FUNCTION_BLOCK FB_CanInterfaceTransport

VAR_INPUT
    bEnable      : BOOL;
END_VAR

VAR_OUTPUT
    xReady       : BOOL;
    xError       : BOOL;
    sErrorText   : STRING(80);
END_VAR

VAR
	TxCanQueue AT%Q* : ST_CanQueue;
	RxCanQueue AT%I* : ST_CanQueue;
END_VAR

END_FUNCTION_BLOCK

(* stored: Version 1.1.0.1
   POU FB_CanInterfaceTransport: Id {351058ca-049c-4ca2-9f12-3a906533c947}, SpecialFunc None *)
